// TIA Portal V20 export
// export: Created 2026-07-16T12:58:45.5217529Z, ExportSetting WithDefaults, DisplayName Totally Integrated Automation Portal, DisplayVersion V20 Update 5, DisplayName TIA Portal Openness, DisplayVersion V20 Update 4, DisplayName TIA Portal Version Control Interface, DisplayVersion V20 Update 5, DisplayName SINAMICS Startdrive Advanced, DisplayVersion V20, DisplayName SINAMICS DCC, DisplayVersion V20, DisplayName SINAMICS Startdrive G130, G150, S120, S150, SINAMICS MV, G220, S200, S210, DisplayVersion V20, DisplayName SINAMICS Startdrive G110M, G120, G120C, G120D, G120P, G115D, DisplayVersion V20, DisplayName STEP 7 Professional, DisplayVersion V20 Update 5, DisplayName STEP 7 Safety, DisplayVersion V20 Update 2, DisplayName WinCC Basic/Comfort/Advanced, DisplayVersion V20 Update 5, DisplayName WinCC Unified, DisplayVersion V20 Update 5
DATA_BLOCK "DB_Output"   // DB2
{ S7_Optimized_Access := 'TRUE' }
VERSION : 0.1
// stored: AutoNumber true, DBAccessibleFromOPCUA true, IsOnlyStoredInLoadMemory false, IsRetainMemResEnabled false, IsWriteProtectedInAS false, MemoryReserve 100
   VAR
      Test : Array[0..18] of Bool;
      SpareDQ : Array[1..7] of Bool;
      Run_Shredder_Fwd : Bool;
      Run_Shredder_Rev : Bool;
      Run_PowerPack : Bool;
      Run_Infeed_Conv : Bool;
      Run_Discharge_Conv : Bool;
      Pusher_Extend : Bool;
      Pusher_Retract : Bool;
      In_Cycle : Bool;
      Enable_Upstream : Bool;
      PreStart_Sounder : Bool;
      Motor_Fault_Reset : Bool;
   END_VAR
BEGIN
END_DATA_BLOCK
